PROGRAM Tsk_MAIN_1ms
VAR


END_VAR

END_PROGRAM

(* stored: Version 1.1.0.1, ProductVersion 3.1.4024.11
   POU Tsk_MAIN_1ms: Id {049e350d-ab9c-4351-80f0-9888af63ceb6}, SpecialFunc None *)
